// TIA Portal V17 export
// export: Created 2022-07-05T09:20:49.0378577Z, ExportSetting WithDefaults, DisplayName Totally Integrated Automation Portal, DisplayVersion V17, DisplayName TIA Portal Openness, DisplayVersion V17, DisplayName TIA Portal Version Control Interface, DisplayVersion V17, DisplayName STEP 7 Professional, DisplayVersion V17, DisplayName STEP 7 Safety, DisplayVersion V17, DisplayName WinCC Advanced, DisplayVersion V17
ORGANIZATION_BLOCK "Main"   // OB1, FBD, ProgramCycle
TITLE = "Main Program Sweep (Cycle)"
{ S7_Optimized_Access := 'TRUE' }
VERSION : 0.1
// stored: AutoNumber true, IsIECCheckEnabled false, SetENOAutomatically false
   VAR_INPUT
      Initial_Call : Bool;   // Initial call of this OB
      Remanence : Bool;   // =True, if remanent data are available
   END_VAR
BEGIN

REGION Network 1: Calling OPC UA client block
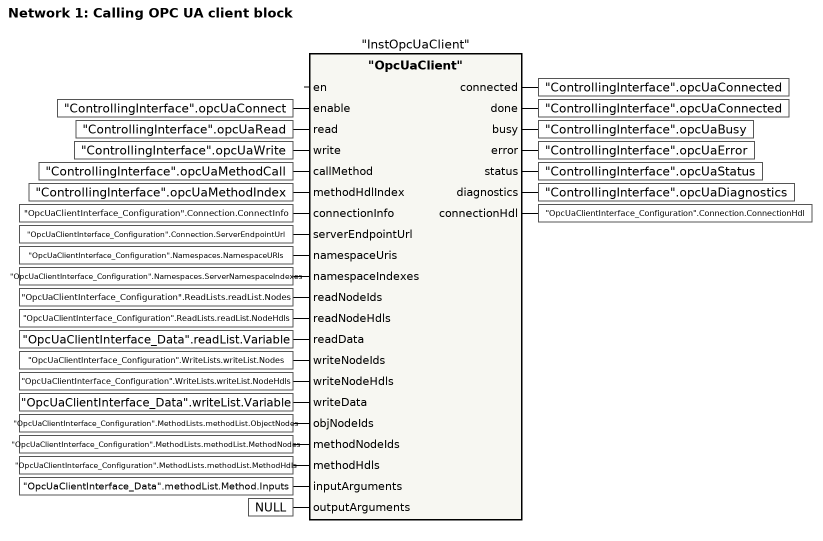
   "InstOpcUaClient"(enable := "ControllingInterface".opcUaConnect,   // "OpcUaClient"
                     read := "ControllingInterface".opcUaRead,
                     write := "ControllingInterface".opcUaWrite,
                     callMethod := "ControllingInterface".opcUaMethodCall,
                     methodHdlIndex := "ControllingInterface".opcUaMethodIndex,
                     connectionInfo := "OpcUaClientInterface_Configuration".Connection.ConnectInfo,
                     serverEndpointUrl := "OpcUaClientInterface_Configuration".Connection.ServerEndpointUrl,
                     namespaceUris := "OpcUaClientInterface_Configuration".Namespaces.NamespaceURIs,
                     namespaceIndexes := "OpcUaClientInterface_Configuration".Namespaces.ServerNamespaceIndexes,
                     readNodeIds := "OpcUaClientInterface_Configuration".ReadLists.readList.Nodes,
                     readNodeHdls := "OpcUaClientInterface_Configuration".ReadLists.readList.NodeHdls,
                     readData := "OpcUaClientInterface_Data".readList.Variable,
                     writeNodeIds := "OpcUaClientInterface_Configuration".WriteLists.writeList.Nodes,
                     writeNodeHdls := "OpcUaClientInterface_Configuration".WriteLists.writeList.NodeHdls,
                     writeData := "OpcUaClientInterface_Data".writeList.Variable,
                     objNodeIds := "OpcUaClientInterface_Configuration".MethodLists.methodList.ObjectNodes,
                     methodNodeIds := "OpcUaClientInterface_Configuration".MethodLists.methodList.MethodNodes,
                     methodHdls := "OpcUaClientInterface_Configuration".MethodLists.methodList.MethodHdls,
                     inputArguments := "OpcUaClientInterface_Data".methodList.Method.Inputs,
                     outputArguments := NULL,
                     connected => "ControllingInterface".opcUaConnected,
                     done => "ControllingInterface".opcUaConnected,
                     busy => "ControllingInterface".opcUaBusy,
                     error => "ControllingInterface".opcUaError,
                     status => "ControllingInterface".opcUaStatus,
                     diagnostics => "ControllingInterface".opcUaDiagnostics,
                     connectionHdl => "OpcUaClientInterface_Configuration".Connection.ConnectionHdl);
END_REGION

REGION Network 2 (SCL)


   "ControllingInterface".new := "ControllingInterface".opcUaDone;
END_REGION
END_ORGANIZATION_BLOCK
